SUBAPPLICATION Uebung_034a3 (* Numeric Value Input auf PWM Ausgang *)
  (* Standard: 61499-2 *)
  (* Version 1.0, 2023-10-23, franz *)
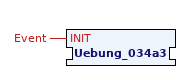
  EVENT_INPUT
    INIT;
  END_EVENT
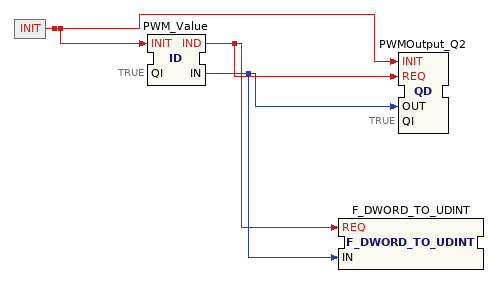
  FBS
    F_DWORD_TO_UDINT : F_DWORD_TO_UDINT;
    PWMOutput_Q2 : QD(QI := TRUE);
    PWM_Value : ID(QI := TRUE);
  END_FBS
  EVENT_CONNECTIONS
    INIT TO PWM_Value.INIT;
    INIT TO PWMOutput_Q2.INIT;
    PWM_Value.IND TO PWMOutput_Q2.REQ;
    PWM_Value.IND TO F_DWORD_TO_UDINT.REQ;
  END_CONNECTIONS
  DATA_CONNECTIONS
    PWM_Value.IN TO F_DWORD_TO_UDINT.IN;
    PWM_Value.IN TO PWMOutput_Q2.OUT;
  END_CONNECTIONS
END_SUBAPPLICATION
